(* IEC 61131-3 sources: controlforge-structured-text/samples/advanced, 3 files *)

(* ---- library.st ---- *)
// Library file with reusable function blocks and functions
// File: samples/advanced/library.st

// Global constants
VAR_GLOBAL CONSTANT
    MAX_TEMPERATURE : REAL := 100.0;
    MIN_TEMPERATURE : REAL := 0.0;
    SYSTEM_VERSION : STRING := 'v2.1.0';
END_VAR

// Utility function for temperature conversion
FUNCTION CelsiusToFahrenheit : REAL
VAR_INPUT
    celsius : REAL;
END_VAR

CelsiusToFahrenheit := celsius * 9.0 / 5.0 + 32.0;

END_FUNCTION

// Advanced PID controller function block
FUNCTION_BLOCK FB_AdvancedPID
VAR_INPUT
    setpoint : REAL;
    processValue : REAL;
    kP : REAL := 1.0;
    kI : REAL := 0.1;
    kD : REAL := 0.01;
    enableIntegral : BOOL := TRUE;
    enableDerivative : BOOL := TRUE;
END_VAR
VAR_OUTPUT
    output : REAL;
    error : REAL;
    saturated : BOOL;
END_VAR
VAR
    integral : REAL;
    lastError : REAL;
    derivative : REAL;
    integralLimit : REAL := 100.0;
END_VAR

// Enhanced PID calculation with saturation handling
error := setpoint - processValue;

// Integral term with windup protection
IF enableIntegral AND NOT saturated THEN
    integral := integral + error;
    integral := LIMIT(integralLimit * -1.0, integral, integralLimit);
END_IF

// Derivative term
IF enableDerivative THEN
    derivative := error - lastError;
END_IF

// PID output calculation
output := kP * error;
IF enableIntegral THEN
    output := output + kI * integral;
END_IF
IF enableDerivative THEN
    output := output + kD * derivative;
END_IF

// Saturation detection
saturated := (output >= 100.0) OR (output <= 0.0);
output := LIMIT(0.0, output, 100.0);

lastError := error;

END_FUNCTION_BLOCK

// Safety monitoring function block
FUNCTION_BLOCK FB_SafetyMonitor
VAR_INPUT
    temperature : REAL;
    pressure : REAL;
    emergencyStop : BOOL;
END_VAR
VAR_OUTPUT
    safetyOK : BOOL;
    alarmActive : BOOL;
    shutdownRequired : BOOL;
END_VAR
VAR
    tempAlarm : BOOL;
    pressureAlarm : BOOL;
END_VAR

// Temperature monitoring
tempAlarm := (temperature > MAX_TEMPERATURE) OR (temperature < MIN_TEMPERATURE);

// Pressure monitoring (assuming max pressure of 10.0 bar)
pressureAlarm := pressure > 10.0;

// Overall safety evaluation
alarmActive := tempAlarm OR pressureAlarm;
shutdownRequired := emergencyStop OR (alarmActive AND (temperature > MAX_TEMPERATURE * 1.1));
safetyOK := NOT alarmActive AND NOT emergencyStop;

END_FUNCTION_BLOCK

(* ---- pid_controller.iecst ---- *)
(* Example IEC Structured Text File *)
FUNCTION_BLOCK FB_PIDController
VAR_INPUT
    SetPoint : REAL;        // Desired value
    ProcessValue : REAL;    // Current value
    Kp : REAL := 1.0;      // Proportional gain
    Ki : REAL := 0.1;      // Integral gain
    Kd : REAL := 0.01;     // Derivative gain
    Enable : BOOL := FALSE; // Enable PID control
END_VAR

VAR_OUTPUT
    Output : REAL;         // Control output
    Error : REAL;         // Current error
END_VAR

VAR
    LastError : REAL;     // Previous error value
    Integral : REAL;      // Integral term
    Derivative : REAL;    // Derivative term
    dt : TIME := T#100ms; // Sample time
END_VAR

// PID Controller Implementation
IF Enable THEN
    // Calculate error
    Error := SetPoint - ProcessValue;

    // Calculate integral term
    Integral := Integral + Error * TIME_TO_REAL(dt);

    // Calculate derivative term
    Derivative := (Error - LastError) / TIME_TO_REAL(dt);

    // Calculate PID output
    Output := Kp * Error + Ki * Integral + Kd * Derivative;

    // Limit output to reasonable range
    IF Output > 100.0 THEN
        Output := 100.0;
    ELSIF Output < -100.0 THEN
        Output := -100.0;
    END_IF

    // Store current error for next cycle
    LastError := Error;
ELSE
    // Reset when disabled
    Output := 0.0;
    Error := 0.0;
    Integral := 0.0;
    LastError := 0.0;
END_IF

END_FUNCTION_BLOCK

(* ---- main-app.st ---- *)
// Main application using library components
// File: samples/advanced/main-app.st
// This file demonstrates cross-file references to library.st

PROGRAM MainApplication
VAR
    // Library function block instances
    temperatureController : FB_AdvancedPID;
    safetySystem : FB_SafetyMonitor;

    // Process variables
    currentTemp : REAL := 25.0;
    currentPressure : REAL := 2.5;
    targetTemp : REAL := 75.0;

    // Control signals
    heaterOutput : REAL;
    emergencyPressed : BOOL := FALSE;

    // Status variables
    systemSafe : BOOL;
    alarmState : BOOL;

    // Converted temperatures for display
    tempInFahrenheit : REAL;

    // Timers
    controlCycleTimer : TON;
    safetyCheckTimer : TON;

    // System info
    version : STRING;
END_VAR

// Initialize system version from global constant
version := SYSTEM_VERSION;

// Convert temperature for display (using library function)
tempInFahrenheit := CelsiusToFahrenheit(currentTemp);

// Temperature control using advanced PID from library
temperatureController(
    setpoint := targetTemp,
    processValue := currentTemp,
    kP := 2.5,
    kI := 0.8,
    kD := 0.15,
    enableIntegral := TRUE,
    enableDerivative := TRUE
);

heaterOutput := temperatureController.output;

// Safety monitoring using library function block
safetySystem(
    temperature := currentTemp,
    pressure := currentPressure,
    emergencyStop := emergencyPressed
);

systemSafe := safetySystem.safetyOK;
alarmState := safetySystem.alarmActive;

// Emergency shutdown if required
IF safetySystem.shutdownRequired THEN
    heaterOutput := 0.0;
    targetTemp := MIN_TEMPERATURE;
END_IF

// Control cycle timing
controlCycleTimer(IN := TRUE, PT := T#100ms);
IF controlCycleTimer.Q THEN
    // Reset timer for next cycle
    controlCycleTimer(IN := FALSE);
END_IF

// Safety check timing
safetyCheckTimer(IN := TRUE, PT := T#50ms);
IF safetyCheckTimer.Q THEN
    // Reset timer for next safety check
    safetyCheckTimer(IN := FALSE);
END_IF

// Temperature bounds checking using global constants
IF targetTemp > MAX_TEMPERATURE THEN
    targetTemp := MAX_TEMPERATURE;
END_IF

IF targetTemp < MIN_TEMPERATURE THEN
    targetTemp := MIN_TEMPERATURE;
END_IF

END_PROGRAM
